TYPE Basic_cycle_Output :
	STRUCT
		Status 	: Basic_cycle_Status_typ;
		Monitor : Basic_cycle_Mon_typ;
		Error 	: Error_Handler_typ;
	END_STRUCT
END_TYPE

(* stored: Version 1.1.0.1, ProductVersion 3.1.4024.3
   DUT Basic_cycle_Output: Id {9830ff4a-e79b-00e3-0e86-15891351ed55} *)
